TYPE EtcSlaveBase_82538BE2 :
STRUCT
END_STRUCT
END_TYPE

(* stored: Version 1.1.0.1, ProductVersion 3.1.4024.9
   DUT EtcSlaveBase_82538BE2: Id {d6b6b4e5-d925-4d4d-b357-2b758ca32e49} *)
